// TIA Portal V19 export
DATA_BLOCK "FP_CM01.GP01"   // DB1001
// stored: AutoNumber false, InstanceOfName FP_Saeure.GP0x, InstanceOfType FB
"FP_Saeure.GP0x"
   // VAR RETAIN
   //    In { ExternalAccessible := 'False'; ExternalVisible := 'False'; ExternalWritable := 'False'} : Struct
   //       NotHalt : Bool;
   //       ext_Freigabe : Bool;
   //       Auto : Bool;
   //       Ein : Bool;
   //       Quitt_FW : Bool;
   //       FU_betriebsbereit : Bool;
   //       FU_Stoerung : Bool;
   //       Niv_TLS : Bool;
   //       Niv_min : Bool;
   //       Niv_max : Bool;
   //       Niv_Uel : Bool;
   //       Frg_Niv_CM05 : Bool;
   //       Leckage_ok : Bool;
   //       SRM_Saugseite_auf : Bool;
   //       SRM_Saugseite_zu : Bool;
   //       SRM_Eingang_Filter_auf : Bool;
   //       SRM_Eingang_Filter_zu : Bool;
   //       SRM_Ausgang_Filter_auf : Bool;
   //       SRM_Ausgang_Filter_zu : Bool;
   //       SRM_Entluften_auf : Bool;
   //       SRM_Entlueften_zu : Bool;
   //       SRM_Eingang_Spülltg_P_auf : Bool;
   //       SRM_Eingang_Spülltg_P_zu : Bool;
   //       SRM_Eingang_Spülltg_F_auf : Bool;
   //       SRM_Eingang_Spülltg_F_zu : Bool;
   //       SRM_Ausgang_Spülltg_auf : Bool;
   //       SRM_Ausgang_Spülltg_zu : Bool;
   //       Sensor_FG_links : Bool;
   //       Sensor_FG_rechts : Bool;
   //       Einhausung_HQ0x_zu : Bool;
   //       GW_p_FP : Bool;
   //       GW_p_FG : Bool;
   //       GW_LF_FP : Bool;
   //       Betriebsart : USInt;
   //       FU_speed : Int;
   //       Druck_Pumpe : Real;
   //       Delta_p_Filter : Real;
   //    END_STRUCT;
   //    Param { ExternalAccessible := 'False'; ExternalVisible := 'False'; ExternalWritable := 'False'} : Struct
   //       SW_Hand : Int;
   //       SW_Auto_AZ : Int;
   //       SW_Auto_aAZ : Int;
   //       Spülzeit_Pumpe : Time;
   //       FG_Zeit_leeren_Saurebecken : Time;
   //       FG_Zeit_leeren_CM05 : Time;
   //       FW_Spülzeit : Time;
   //       FW_Wartezeit : Time;
   //       FW_Zeit_fuellen : Time;
   //       DT_Druckaufbau : Time;
   //       DT_Testzeit_Pumpe : Time;
   //       DT_Testzeit_Filter : Time;
   //       SW_Drucktest_Pumpe : Real;
   //       SW_Drucktest_Filter : Real;
   //       WarnGr_FW : Real;
   //       Wechsel_FW : Real;
   //       Name_Pumpe : String[12];
   //       Name_Filter : String[12];
   //    END_STRUCT;
   //    Zst { ExternalAccessible := 'False'; ExternalVisible := 'False'; ExternalWritable := 'False'} : Struct
   //       Status_GP0x : USInt;
   //       Status_FW : USInt;
   //       Status_DT_Pumpe : USInt;
   //       Status_DT_Filter : USInt;
   //       Restzeit_Spülen_Pumpe : Time;
   //       Restzeit_Filter : Time;
   //       Restzeit_DT : Time;
   //       Spuelen_Pumpe : Bool;
   //       Spuelen_Filter : Bool;
   //       Spuelen_aktiv : Bool;
   //       Drucktest_aktiv : Bool;
   //       Filtern : Bool;
   //       Zeit_laeuft : Bool;
   //       Drucktest_Pu_ok : Bool;
   //       Drucktest_Filter_ok : Bool;
   //       Bedienung_erlaubt : Bool;
   //       speed : Int;
   //    END_STRUCT;
   //    Mld { ExternalAccessible := 'False'; ExternalVisible := 'False'; ExternalWritable := 'False'} : Struct
   //       Leckage : Bool;
   //       GW_p_FP : Bool;
   //       GW_LF_FP : Bool;
   //       GW_p_FG : Bool;
   //       FG_links_nicht_zu : Bool;
   //       FG_rechts_nicht_zu : Bool;
   //       Einhausung_nicht_zu : Bool;
   //       FU_nicht_bereit : Bool;
   //       FU_Stoerung : Bool;
   //       FG_Spülen_Ende : Bool;
   //       n_Auto : Bool;
   //       TO_Druckaufbau : Bool;
   //       Drucktest_Pumpe_ok : Bool;
   //       Drucktest_Pumpe_Fehler : Bool;
   //       Pu_Spuelen_Fertig : Bool;
   //       Drucktest_Filter_ok : Bool;
   //       Drucktest_Filter_Fehler : Bool;
   //       Drucktest_Filter_erfordert : Bool;
   //       Filterbeutel_Wechsel_Vorwarngrenze : Bool;
   //       Filterbeutel_Wechsel_notwendig : Bool;
   //    END_STRUCT;
   //    Out { ExternalAccessible := 'False'; ExternalVisible := 'False'; ExternalWritable := 'False'} : Struct
   //       GP0x_Ein : Bool;
   //       Ventil_Saugseite : Bool;
   //       Ventil_Eingang_Filter : Bool;
   //       Ventil_Ausgang_Filter : Bool;
   //       Ventil_Entlueften : Bool;
   //       Spülventil_P_Eingang : Bool;
   //       Spülventil_F_Eingang : Bool;
   //       Spülventil_Ausgang : Bool;
   //       Soll_speed : Int;
   //    END_STRUCT;
   // END_VAR
   // VAR
   //    IEC_Timer { ExternalAccessible := 'False'; ExternalVisible := 'False'; ExternalWritable := 'False'} : Struct
   //       Spülen_Pumpe { S7_SetPoint := 'True'} : TP_TIME;
   //       Filterwechsel { S7_SetPoint := 'True'} : TP_TIME;
   //       GW_p { S7_SetPoint := 'True'} : TON_TIME;
   //       Drucktest { S7_SetPoint := 'True'} : TP_TIME;
   //       TO_Druckaufbau { S7_SetPoint := 'True'} : TON_TIME;
   //       Verz_Ueberdruck { S7_SetPoint := 'True'} : TON_TIME;
   //       Spülventil_Ausgang { S7_SetPoint := 'True'} : TOF_TIME;
   //    END_STRUCT;
   //    R_TRIG_Hand_EIN { ExternalAccessible := 'False'; ExternalVisible := 'False'; ExternalWritable := 'False'} : R_TRIG;
   // END_VAR
BEGIN
END_DATA_BLOCK
